SUBAPPLICATION AUS_AUI_MUX_3_VAL (* 3-Wege-Multiplexer fuer AUS-Werte mit 3 internen initval_AUS und AUI_MUX_3 / AUS_AUI_MUX_3. Schaltet per Event-Input (EI1, EI2, EI3) zwischen val1, val2, val3 um. *)
  (* Standard: 61499-2; Description: Copyright (c) 2026 Meisterschulen am Ostbahnhof This program and the accompanying materials are made available under the terms of the Eclipse Public License 2.0 which is available at https://www.eclipse.org/legal/epl-2.0/ SPDX-License-Identifier: EPL-2.0 *)
  (* Version 1.0, 2026-09-10, Franz Höpfinger, Meisterschulen am Ostbahnhof, initial implementation *)
  PACKAGE MyLib::sys;
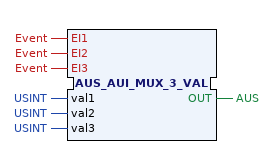
  EVENT_INPUT
    EI1; (* Event zur Auswahl von val1 *)
    EI2; (* Event zur Auswahl von val2 *)
    EI3; (* Event zur Auswahl von val3 *)
  END_EVENT
  VAR_INPUT
    val1 : USINT; (* Initialer Ausgabewert bei EI1 *)
    val2 : USINT; (* Initialer Ausgabewert bei EI2 *)
    val3 : USINT; (* Initialer Ausgabewert bei EI3 *)
  END_VAR
  PLUGS
    OUT : adapter::types::unidirectional::AUS; (* Ausgewaehlter AUS-Adapter Output *)
  END_PLUGS
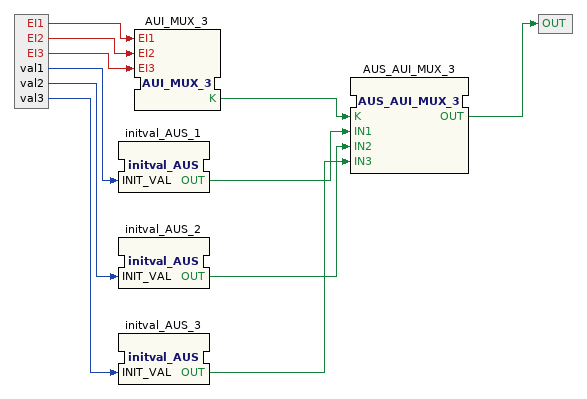
  FBS
    AUI_MUX_3 : adapter::events::unidirectional::AUI_MUX_3;
    AUS_AUI_MUX_3 : adapter::selection::unidirectional::AUS_AUI_MUX_3;
    initval_AUS_1 : adapter::types::unidirectional::AUS::initval::initval_AUS;
    initval_AUS_2 : adapter::types::unidirectional::AUS::initval::initval_AUS;
    initval_AUS_3 : adapter::types::unidirectional::AUS::initval::initval_AUS;
  END_FBS
  EVENT_CONNECTIONS
    EI1 TO AUI_MUX_3.EI1;
    EI2 TO AUI_MUX_3.EI2;
    EI3 TO AUI_MUX_3.EI3;
  END_CONNECTIONS
  DATA_CONNECTIONS
    val1 TO initval_AUS_1.INIT_VAL;
    val2 TO initval_AUS_2.INIT_VAL;
    val3 TO initval_AUS_3.INIT_VAL;
  END_CONNECTIONS
  ADAPTER_CONNECTIONS
    AUI_MUX_3.K TO AUS_AUI_MUX_3.K;
    initval_AUS_1.OUT TO AUS_AUI_MUX_3.IN1;
    initval_AUS_2.OUT TO AUS_AUI_MUX_3.IN2;
    initval_AUS_3.OUT TO AUS_AUI_MUX_3.IN3;
    AUS_AUI_MUX_3.OUT TO OUT;
  END_CONNECTIONS
END_SUBAPPLICATION
